TYPE T_ACTUATOR_CTRL :
STRUCT
	nCommand:		DINT	:= E_ACTUATOR_COMMAND.NONE;	(* See E_ACTUATOR_COMMAND *)
	bExecute:		BOOL;
	
END_STRUCT
END_TYPE

(* stored: Version 1.1.0.1, ProductVersion 3.1.4024.3
   DUT T_ACTUATOR_CTRL: Id {17405076-e76e-47ad-8e66-f8b937714847} *)
